(* IEC 61131-3 sources: json/src/Elements/Numbers, 11 files *)

(* ---- BaseJsonNumber.st ---- *)
USING System.Strings;

NAMESPACE Simatic.Ax.Json
    {axcode:docs-v0:@simatic-ax/json:../README.md}
    CLASS BaseJsonNumber EXTENDS AbstractJsonElement

        METHOD PROTECTED OVERRIDE ToStringHelper : STRING
            VAR_INPUT
                valueAsString : STRING;
            END_VAR
            VAR_TEMP
                _str : STRING;
            END_VAR
            _str := Concat('"', Key, '": ', valueAsString);
            ToStringHelper := _str;
        END_METHOD

        METHOD PUBLIC OVERRIDE ToString : STRING
            ;
        END_METHOD

        METHOD PUBLIC OVERRIDE Serialize : BOOL
            VAR_INPUT
                doc : REF_TO JsonDocument;
            END_VAR
            THIS.SerializeHelper(doc, THIS.ToString());
            Serialize := FALSE;
        END_METHOD
    END_CLASS
END_NAMESPACE

(* ---- DoubleInt.st ---- *)
USING Simatic.Ax.Conversion;

NAMESPACE Simatic.Ax.Json
    CLASS JsonDoubleInt EXTENDS JsonNumber
        VAR PUBLIC
            value : DINT;
        END_VAR

        METHOD PUBLIC OVERRIDE ToString : STRING
            ToString := THIS.ToStringHelper(Integer.ToString(value := value));
        END_METHOD
    END_CLASS
END_NAMESPACE

(* ---- JsonDInt.st ---- *)
USING Simatic.Ax.Conversion;

NAMESPACE Simatic.Ax.Json
    CLASS FINAL JsonDInt EXTENDS BaseJsonNumber
        VAR PUBLIC
            Value : DINT;
        END_VAR

        METHOD PUBLIC OVERRIDE ToString : STRING
            ToString := THIS.ToStringHelper(Integer.ToString(value := Value));
        END_METHOD

    END_CLASS
END_NAMESPACE

(* ---- JsonDoubleInt.st ---- *)
USING Simatic.Ax.Conversion;

NAMESPACE Simatic.Ax.Json
    CLASS JsonDoubleInt EXTENDS JsonNumber
        VAR PUBLIC
            Value : DINT;
        END_VAR

        METHOD PUBLIC OVERRIDE ToString : STRING
            ToString := THIS.ToStringHelper(Integer.ToString(value := Value));
        END_METHOD

        METHOD PUBLIC OVERRIDE Serialize : BOOL
            VAR_INPUT
                doc : REF_TO JsonDocument;
            END_VAR
            THIS.SerializeHelper(doc, THIS.ToString());
            Serialize := FALSE;
        END_METHOD
    END_CLASS
END_NAMESPACE

(* ---- JsonInt.st ---- *)
USING Simatic.Ax.Conversion;

NAMESPACE Simatic.Ax.Json
    CLASS JsonInt EXTENDS JsonNumber
        VAR PUBLIC
            value : INT;
        END_VAR

        METHOD PUBLIC OVERRIDE ToString : STRING
            ToString := THIS.ToStringHelper(Integer.ToString(value := value));
        END_METHOD
    END_CLASS
END_NAMESPACE

(* ---- JsonLInt.st ---- *)
USING Simatic.Ax.Conversion;

NAMESPACE Simatic.Ax.Json
    CLASS JsonLInt EXTENDS BaseJsonNumber
        VAR PUBLIC
            Value : LINT;
        END_VAR

        METHOD PUBLIC OVERRIDE ToString : STRING
            ToString := THIS.ToStringHelper(Integer.ToString(value := Value));
        END_METHOD

    END_CLASS
END_NAMESPACE

(* ---- JsonLongInt.st ---- *)
USING Simatic.Ax.Conversion;

NAMESPACE Simatic.Ax.Json
    CLASS JsonLongInt EXTENDS JsonNumber
        VAR PUBLIC
            Value : LINT;
        END_VAR

        METHOD PUBLIC OVERRIDE ToString : STRING
            ToString := THIS.ToStringHelper(Integer.ToString(value := Value));
        END_METHOD

        METHOD PUBLIC OVERRIDE Serialize : BOOL
            VAR_INPUT
                doc : REF_TO JsonDocument;
            END_VAR
            THIS.SerializeHelper(doc, THIS.ToString());
            Serialize := FALSE;
        END_METHOD

    END_CLASS
END_NAMESPACE

(* ---- JsonNumber.st ---- *)
USING System.Strings;

NAMESPACE Simatic.Ax.Json
    CLASS JsonNumber EXTENDS AbstractJsonElement

        METHOD PROTECTED OVERRIDE ToStringHelper : STRING
            VAR_INPUT
                valueAsString : STRING;
            END_VAR
            VAR_TEMP
                _str : STRING;
            END_VAR
            _str := Concat('"', key, '": ', valueAsString);
            ToStringHelper := _str;
        END_METHOD

        METHOD PUBLIC OVERRIDE ToString : STRING
            ;
        END_METHOD
    END_CLASS
END_NAMESPACE

(* ---- JsonSint.st ---- *)
USING Simatic.Ax.Conversion;

NAMESPACE Simatic.Ax.Json
    CLASS JsonUSInt EXTENDS BaseJsonNumber
        VAR PUBLIC
            Value : USINT;
        END_VAR

        METHOD PUBLIC OVERRIDE ToString : STRING
            ToString := THIS.ToStringHelper(Integer.ToString(value := Value));
        END_METHOD

    END_CLASS
END_NAMESPACE

(* ---- JsonUint.st ---- *)
USING Simatic.Ax.Conversion;

NAMESPACE Simatic.Ax.Json
    CLASS JsonSInt EXTENDS JsonNumber
        VAR PUBLIC
            Value : SINT;
        END_VAR

        METHOD PUBLIC OVERRIDE ToString : STRING
            ToString := THIS.ToStringHelper(Integer.ToString(value := Value));
        END_METHOD

    END_CLASS
END_NAMESPACE

(* ---- JsonUSint.st ---- *)
USING Simatic.Ax.Conversion;

NAMESPACE Simatic.Ax.Json
    CLASS FINAL JsonUSInt EXTENDS BaseJsonNumber
        VAR PUBLIC
            Value : USINT;
        END_VAR

        METHOD PUBLIC OVERRIDE ToString : STRING
            ToString := THIS.ToStringHelper(Integer.ToString(value := Value));
        END_METHOD

    END_CLASS
END_NAMESPACE
